// TIA Portal project "Clase 6 SCL" (V14)

(* hardware
DEVICE "S7-1200 station_1"  S7-1200 Station
   slot 0: "Rack_0"  S7-1200 Rack  Rack  V1.0
   slot 1: "PLC_1"  CPU 1214C DC/DC/DC  6ES7 214-1AG40-0XB0  V4.2
*)

// ===== PLC "PLC_1"  CPU 1214C DC/DC/DC =====

VAR_GLOBAL   // PLC tag table "Salidas"
   "Luz Verde Parking Accesible" AT %Q0.0 : Bool;
   "Luz Roja Parking Completo" AT %Q0.1 : Bool;
   "Abrir Barrera Entrada (KM1)" AT %Q0.2 : Bool;
   "Cerrar Barrera Entrada (KM2)" AT %Q0.3 : Bool;
   "Abrir Barrera Salida (KM3)" AT %Q0.4 : Bool;
   "Cerrar Barrera Salida (KM4)" AT %Q0.5 : Bool;
   "SalidaTempImpulso" AT %Q0.6 : Bool;
   "SalidaTempAcumulativo" AT %Q0.7 : Bool;
END_VAR

VAR_GLOBAL   // PLC tag table "Entradas"
   "Rele termico" AT %I0.0 : Bool;
   "Pulsador Start" AT %I0.1 : Bool;
   "Pulsador Stop" AT %I0.2 : Bool;
   "Seta Emergencia" AT %I0.3 : Bool;
   "Sensor Entrada" AT %I0.4 : Bool;
   "Sensor Salida" AT %I0.5 : Bool;
   "FC. Barrera Entrada Abierta" AT %I0.6 : Bool;
   "FC. Barrera Entrada Cerrada" AT %I0.7 : Bool;
   "FC. Barrera Salida Abierta" AT %I1.0 : Bool;
   "FC. Barrara Salida Cerrada" AT %I1.1 : Bool;
   "Pulsador Abrir Barrera Entrada" AT %I1.2 : Bool;
   "Pulsador Abrir Barrera Salida" AT %I1.3 : Bool;
   "PulsadorReset" AT %I1.4 : Bool;
END_VAR

DATA_BLOCK "var"   // DB1
{ S7_Optimized_Access := 'TRUE' }
VERSION : 0.1
   VAR
      General : Struct
         Sistemas : Struct
            "Sistema OK" : Bool;
            Inicial : Bool;
            "Parking Disponible" : Bool;
            "Parking Completo" : Bool;
            "Estado Parking" : WString;
            DTL_LOC : DTL;
            DTL_ENTRADA : DTL;
            RET_VAL_LOC : Int;
            TIEMPO_TOTAL : Time_Of_Day;
         END_STRUCT;
         "Barrera Entrada" : Struct
            "Act. Subida Barrera" : Bool;
            "Act. Bajada Barrera" : Bool;
         END_STRUCT;
         "Barrera Salida" : Struct
            "Act. Subida Barrera" : Bool;
            "Act. Bajada Barrera" : Bool;
         END_STRUCT;
      END_STRUCT;
      "Cont/Temp" : Struct
         Contadores : Struct
            ResetCount : Bool;
            "Contaje Ascendente" : Bool;
            "Contaje Descendente" : Bool;
            CTUD : IEC_COUNTER;
         END_STRUCT;
         Temporizadores : Struct
            "Act.TempSalida" : Bool;
            "Act.TempEntrada" : Bool;
            TempSalidaOk : Bool;
            TempEntradaOk : Bool;
            TempTimeEntrada : Time;
            TempTimeSalida : Time;
            TempTimeImpulso : Time;
            TempTimeAcumulativo : Time;
            TemporizadorSalida : IEC_TIMER;
            TemporizadorEntrada : IEC_TIMER;
            TemporizadorImpulso : IEC_TIMER;
            TemporizadorAcumulativo : IEC_TIMER;
         END_STRUCT;
      END_STRUCT;
   END_VAR
BEGIN
END_DATA_BLOCK

FUNCTION "(1) Condicionales" : Void   // FC1, SCL
{ S7_Optimized_Access := 'TRUE' }
VERSION : 0.1
BEGIN
   (*************************************************************************************************************
                                                 Programa plc: Función Condicionales
   **************************************************************************************************************

   *    Proyecto: Clase 5 de programación en lenguaje SCL para TIA PORTAL (TEMPORIZADORES)
   *    Equipo: Automata Plc Siemens S7-1200
   *    Designer: Jesús Alguacil
   *    Responsable:
   *    Fecha: 20/08/2021

   **************************************************************************************************************)

   REGION ESTRUCTURA DEL BLOQUE CONDICIONALES
       REGION Condicional CASE
           CASE "var"."Cont/Temp".Contadores.CTUD.CV OF
               0..9:
                   IF "var".General.Sistemas."Sistema OK" THEN
                       "var".General.Sistemas."Parking Disponible" := true;
                       "var".General.Sistemas."Parking Completo" := false;
                       "var".General.Sistemas."Estado Parking" := WSTRING#'Parking Disponible';
                       REGION Condicionante Descendente
                           IF "var"."Cont/Temp".Contadores.CTUD.CV = 0 THEN
                               "var".General.Sistemas.Inicial := true;
                           ELSE
                               "var".General.Sistemas.Inicial := false;
                           END_IF;
                       END_REGION
                   END_IF;
               10:
                   IF "var".General.Sistemas."Sistema OK" THEN
                       "var".General.Sistemas."Parking Completo" := true;
                       "var".General.Sistemas."Parking Disponible" := false;
                       "var".General.Sistemas."Estado Parking" := WSTRING#'Parking Completo';
                   END_IF;
           END_CASE;
       END_REGION

       REGION Condicionales de los temporizadores
           REGION Temporizador de entrada
               IF "var"."Cont/Temp".Contadores."Contaje Ascendente" THEN
                   "var"."Cont/Temp".Temporizadores."Act.TempEntrada" := true;
               ELSIF
                   "var"."Cont/Temp".Temporizadores.TempEntradaOk THEN
                   "var"."Cont/Temp".Temporizadores."Act.TempEntrada" := false;
               END_IF;
           END_REGION

           REGION Temporizador de salida
               IF "var"."Cont/Temp".Contadores."Contaje Descendente" THEN
                   "var"."Cont/Temp".Temporizadores."Act.TempSalida" := true;
               ELSIF
                   "var"."Cont/Temp".Temporizadores.TempSalidaOk THEN
                   "var"."Cont/Temp".Temporizadores."Act.TempSalida" := false;
               END_IF;
           END_REGION
       END_REGION

       REGION Activación de las barreras del parking
           REGION Barrera de Entrada al Parking
               REGION Subida
                   IF "var".General.Sistemas."Sistema OK" AND "var".General.Sistemas."Parking Disponible" AND "Pulsador Abrir Barrera Entrada" THEN
                       "var".General."Barrera Entrada"."Act. Subida Barrera" := true;
                   ELSIF
                       "var".General.Sistemas."Sistema OK" AND "FC. Barrera Entrada Abierta" AND NOT "FC. Barrera Entrada Cerrada" THEN
                       "var".General."Barrera Entrada"."Act. Subida Barrera" := false;
                   END_IF;

               END_REGION
               REGION Bajada
                   IF "var".General.Sistemas."Sistema OK" AND "FC. Barrera Entrada Abierta" AND "var"."Cont/Temp".Temporizadores.TempEntradaOk THEN
                       "var".General."Barrera Entrada"."Act. Bajada Barrera" := true;
                   ELSIF // parada de la bajada 
                       "var".General.Sistemas."Sistema OK" AND NOT "FC. Barrera Entrada Abierta" AND "FC. Barrera Entrada Cerrada" THEN
                       "var".General."Barrera Entrada"."Act. Bajada Barrera" := false;
                   END_IF;
               END_REGION
           END_REGION

           REGION Barrera de Salida del Parking
               REGION Subida
                   IF "var".General.Sistemas."Sistema OK" AND "Pulsador Abrir Barrera Salida" THEN
                       "var".General."Barrera Salida"."Act. Subida Barrera" := true;
                   ELSIF
                       "var".General.Sistemas."Sistema OK" AND "FC. Barrera Salida Abierta" AND NOT "FC. Barrara Salida Cerrada" THEN
                       "var".General."Barrera Salida"."Act. Subida Barrera" := false;
                   END_IF;
               END_REGION
               REGION Bajada
                   IF "var".General.Sistemas."Sistema OK" AND "FC. Barrera Salida Abierta" AND "var"."Cont/Temp".Temporizadores.TempSalidaOk THEN
                       "var".General."Barrera Salida"."Act. Bajada Barrera" := true;
                   ELSIF // parada de la bajada
                       "var".General.Sistemas."Sistema OK" AND NOT "FC. Barrera Salida Abierta" AND "FC. Barrara Salida Cerrada" THEN
                       "var".General."Barrera Salida"."Act. Bajada Barrera" := false;
                   END_IF;
               END_REGION
           END_REGION
       END_REGION
   END_REGION

   // END BLOCK
END_FUNCTION

FUNCTION "(2) Contadores/Temporizadores" : Void   // FC2, SCL
{ S7_Optimized_Access := 'TRUE' }
VERSION : 0.1
BEGIN
   (*************************************************************************************************************
                                                 Programa plc: Función Contadores/Temporizadores
   **************************************************************************************************************

   *    Proyecto: Clase 6 de programación en lenguaje SCL para TIA PORTAL (TEMPORIZADORES)
   *    Equipo: Automata Plc Siemens S7-1200
   *    Designer: Jesús Alguacil
   *    Responsable:
   *    Fecha: 03/09/2021

   **************************************************************************************************************)

   Region ESTRUCTURA DEL BLOQUE CONTADORES/TEMPORIZADORES
       Region Activación de los flancos para el contador del parking
           Region Flanco "Descendente" para el contaje ascendente de vehiculos en el parking
               "F_TRIG_INCREMENTO"(CLK:="Sensor Entrada",
                                   Q=>"var"."Cont/Temp".Contadores."Contaje Ascendente");
           END_REGION
           Region Flanco "Descendente" para el contaje descendente de vehiculos en el parking
               "F_TRIG_DECREMENTO"(CLK:="Sensor Salida",
                                   Q=>"var"."Cont/Temp".Contadores."Contaje Descendente");
           END_REGION
       END_REGION

       Region Contador de vehiculos para el parking
           "var"."Cont/Temp".Contadores.CTUD.CTUD(CU:="var"."Cont/Temp".Contadores."Contaje Ascendente" AND NOT "var".General.Sistemas."Parking Completo",
                                                  CD:="var"."Cont/Temp".Contadores."Contaje Descendente" AND NOT "var".General.Sistemas.Inicial,
                                                  R:="var"."Cont/Temp".Contadores.ResetCount,
                                                  PV:="var"."Cont/Temp".Contadores.CTUD.PV,
                                                  CV=>"var"."Cont/Temp".Contadores.CTUD.CV);
       END_REGION

       Region Temporizadores
           Region Temporizador para la bajada de la barrera de entrada
               "var"."Cont/Temp".Temporizadores.TemporizadorEntrada.TON(IN := "var"."Cont/Temp".Temporizadores."Act.TempEntrada",
                                                                        PT := T#10s,
                                                                        Q => "var"."Cont/Temp".Temporizadores.TempEntradaOk,
                                                                        ET => "var"."Cont/Temp".Temporizadores.TempTimeEntrada);
           END_REGION
           Region Temporizador para la bajada de la barrera de salida
               "var"."Cont/Temp".Temporizadores.TemporizadorSalida.TON(IN:="var"."Cont/Temp".Temporizadores."Act.TempSalida",
                                                                       PT:=T#5s,
                                                                       Q=>"var"."Cont/Temp".Temporizadores.TempSalidaOk,
                                                                       ET=>"var"."Cont/Temp".Temporizadores.TempTimeSalida);
           END_REGION
           Region Temporizador de impulso mediante flanco
               "var"."Cont/Temp".Temporizadores.TemporizadorImpulso.TP(IN := "var"."Cont/Temp".Contadores."Contaje Ascendente",
                                                                       PT := T#5s,
                                                                       Q => "SalidaTempImpulso",
                                                                       ET => "var"."Cont/Temp".Temporizadores.TempTimeImpulso);
           END_REGION
           Region Temporizador Acumulativo
               "var"."Cont/Temp".Temporizadores.TemporizadorAcumulativo.TONR(IN := "Pulsador Start",
                                                                             PT := T#30s,
                                                                             Q => "SalidaTempAcumulativo",
                                                                             ET => "var"."Cont/Temp".Temporizadores.TempTimeAcumulativo);


           END_REGION

           Region
               "var".General.Sistemas.RET_VAL_LOC := RD_LOC_T("var".General.Sistemas.DTL_LOC);
               "var".General.Sistemas.TIEMPO_TOTAL := T_DIFF(IN1 := "var".General.Sistemas.DTL_LOC, IN2 := "var".General.Sistemas.DTL_ENTRADA);
           END_REGION
       END_REGION
       Region Asignación del valor PV al contaje
           "var"."Cont/Temp".Contadores.CTUD.PV := 10;
       END_REGION
   END_REGION

   // END BLOCK
END_FUNCTION

FUNCTION "(3) Salidas" : Void   // FC3, SCL
{ S7_Optimized_Access := 'TRUE' }
VERSION : 0.1
BEGIN
   (*************************************************************************************************************
                                                 Programa plc: Función Salidas
   **************************************************************************************************************

   *    Proyecto: Clase 5 de programación en lenguaje SCL para TIA PORTAL (TEMPORIZADORES)
   *    Equipo: Automata Plc Siemens S7-1200
   *    Designer: Jesús Alguacil
   *    Responsable:
   *    Fecha: 20/08/2021

   **************************************************************************************************************)

   REGION ESTRUCTURA DEL BLOQUE SALIDAS
       // SALIDA Q0.0
       "Luz Verde Parking Accesible" := "var".General.Sistemas."Parking Disponible";

       // SALIDA Q0.1
       "Luz Roja Parking Completo" := "var".General.Sistemas."Parking Completo";

       // SALIDA Q0.2
       "Abrir Barrera Entrada (KM1)" := "var".General."Barrera Entrada"."Act. Subida Barrera";

       // SALIDA Q0.3
       "Cerrar Barrera Entrada (KM2)" := "var".General."Barrera Entrada"."Act. Bajada Barrera";

       // SALIDA Q0.4
       "Abrir Barrera Salida (KM3)" := "var".General."Barrera Salida"."Act. Subida Barrera";

       // SALIDA Q0.5
       "Cerrar Barrera Salida (KM4)" := "var".General."Barrera Salida"."Act. Bajada Barrera";
   END_REGION

   // END BLOCK
END_FUNCTION

ORGANIZATION_BLOCK "Main"   // OB1, SCL, ProgramCycle
TITLE = "Main Program Sweep (Cycle)"
{ S7_Optimized_Access := 'TRUE' }
VERSION : 0.1
   VAR_INPUT
      Initial_Call : Bool;   // Initial call of this OB
      Remanence : Bool;   // =True, if remanent data are available
   END_VAR
BEGIN
   (*************************************************************************************************************
                                                 Programa plc: Main
   **************************************************************************************************************

   *    Proyecto: Clase 4 de programación en lenguaje SCL para TIA PORTAL (INSTRUCCIÓN CASE/IF)
   *    Equipo: Automata Plc Siemens S7-1200
   *    Designer: Jesús Alguacil
   *    Responsable:
   *    Fecha: 03/06/2021 (Fecha prevista terminación viernes 04/06/2021)

   **************************************************************************************************************)

   REGION ESTRUCTURA DEL BLOQUE MAIN
       REGION Funciones (Llamamos a los bloques de función para su ejecución)
           "(1) Condicionales"();
           "(2) Contadores/Temporizadores"();
           "(3) Salidas"();
       END_REGION

       REGION Señales de seguridad
           "var".General.Sistemas."Sistema OK" := "Rele termico" AND "Seta Emergencia";
           "var"."Cont/Temp".Contadores.ResetCount := NOT "Pulsador Stop";
       END_REGION
   END_REGION

   // END BLOCK
END_ORGANIZATION_BLOCK